// TIA Portal V20 export
TYPE "Size"
// stored: Access Published, Namespace LER
   STRUCT
      Anode : Struct
         thickness : LReal;
         width : LReal;
         length : LReal;
      END_STRUCT;
      Cathode : Struct
         thickness : LReal;
         width : LReal;
         length : LReal;
      END_STRUCT;
      Offset : LReal;
   END_STRUCT;
END_TYPE
